TYPE
    PiperModuleInternal :
    STRUCT
        machine : REFERENCE TO Piper;
        context : IPluginRunner;
        registered : BOOL;
        response : RESPONSE_STATE;
        requestSubstate : ULINT;
        previousSubstate : ULINT;
        previousSubstateAsync : ULINT;
        skipsSync : PiperImplements;
        skipsAsync : PiperImplements;
        requestNumber : DINT;
    END_STRUCT
END_TYPE

(* stored: Version 1.1.0.1
   DUT PiperModuleInternal: Id {44cb28c5-3604-437e-8c8d-62be209a7d26} *)
